ABB RobotStudio station: Assistenzsystem für Verpressung.rsstnx

Station Assistenzsystem für Verpressung (saved by RobotStudio 22.3.10190.2)
Controller IRB14000
  mechanical unit ROB_R: IRB14000_0.5_0.5_R, 6 joints, base frame (0, 0, 0) mm
  mechanical unit ROB_R_7: IRB14000_0.5_0.5_R, 1 joints, base frame (0, 0, 0) mm
  mechanical unit ROB_L: IRB14000_0.5_0.5_L, 6 joints, base frame (0, 0, 0) mm
  mechanical unit ROB_L_7: IRB14000_0.5_0.5_L, 1 joints, base frame (0, 0, 0) mm
Layout (positions relative to the parent item):
  - IRB14000_0.5_0.5 [mechanism, from Robots\IRB14000_0.5_0.5__01.rslib] at (0, 0, 0) mm
  - IRB14000_0.5_0.5_R [mechanism, from Robots\IRB14000_0.5_0.5__01.rslib] at (0, 0, 0) mm; joint values [0.3584, -1.8727, -2.4697, 0.5522, 0.721, 0.9332, -0.6165] (rad or m)
  - IRB14000_0.5_0.5_L [mechanism, from Robots\IRB14000_0.5_0.5__01.rslib] at (0, 0, 0) mm; joint values [-0.3584, -1.8727, 2.4697, 0.5522, -0.721, 0.9332, 0.6165] (rad or m)
  - Smart_Gripper_Servo_Fingers_R [mechanism, from Tools\ABB_Smart_Gripper_Servo_Fingers.rslib] at (-9.58, -182.61, 198.63) mm, rotated rx 179.34 ry -63.63 rz 15.45 deg; joint values [0] (rad or m)
  - Smart_Gripper_Servo_Fingers_L [mechanism, from Tools\ABB_Smart_Gripper_Servo_Fingers.rslib] at (-9.58, 182.61, 198.63) mm, rotated rx -179.34 ry -63.63 rz -15.45 deg; joint values [0] (rad or m)
Attachment: Smart_Gripper_Servo_Fingers_R is attached to IRB14000_0.5_0.5_R / Link7
Attachment: Smart_Gripper_Servo_Fingers_L is attached to IRB14000_0.5_0.5_L / Link7
Targets, tools, work objects and paths stored in the station, written as RAPID:
! task T_ROB_R
MODULE CalibData
  PERS tooldata Servo:=[TRUE,[[0,0,114.2],[1,0,0,0]],[0.215,[8.7,12.3,49.2],[1,0,0,0],0.00021,0.00024,0.00009]];
ENDMODULE

! task T_ROB_L
MODULE CalibData
  PERS tooldata Servo:=[TRUE,[[0,0,114.2],[1,0,0,0]],[0.215,[8.7,12.3,49.2],[1,0,0,0],0.00021,0.00024,0.00009]];
ENDMODULE

